{attribute addProperty BoxType "EL3773-0000-0018"}
{attribute addProperty Id "U3_SamplesAT %I*ARRAY [1..10] OF INT16020"}
{attribute addProperty CRC "3234393355"}
{attribute addProperty SizeInBites "160"}
{attribute addProperty SizeInBytes "20"}
TYPE L3_Voltage_Samples_C0C8ED0B :
STRUCT
	{attribute addProperty Name "U3_Samples"}
	U3_Samples AT %I* : ARRAY [1..10] OF INT;
END_STRUCT
END_TYPE

(* stored: Version 1.2.0.0, ProductVersion 3.1.4024.9
   DUT L3_Voltage_Samples_C0C8ED0B: Id {acc3afca-acff-40ba-bfe7-e36d0093a411} *)
